TYPE EM_Transport_SIM :
STRUCT
	Stopping_SC	: BOOL;
END_STRUCT
END_TYPE

(* stored: Version 1.1.0.1, ProductVersion 3.1.4024.12
   DUT EM_Transport_SIM: Id {8d300077-1d88-4620-8ced-a9ca53cd20c9} *)
